KUKA KRL data list: Up22.dat

&ACCESS RVO1
&REL 340
&COMMENT VW380 HO_Behaelter_rechts
&PARAM EDITMASK = Up999[1-999]
&PARAM TEMPLATE = C:\KRC\Roboter\Template\upvorgabe
&PARAM TPVW_VERSION = 8.3.18
&PARAM DISKPATH = UPs
DEFDAT UP22
; FOLD ;%{H} %MKUKATPVW
; ENDFOLD
; interface to basic routines
 EXT  BAS (BAS_COMMAND  :IN,REAL  :IN )
; interface to VW-standard routines
EXT VW (VW_COMMAND:IN, BOOL: IN, REAL:IN, REAL:IN, REAL:IN, REAL:IN, BOOL :IN, E6POS :IN )
; interface to VW_USER - Call
EXT  VW_USER (VW_USER_CMD :IN,INT :IN,REAL  :IN,REAL  :IN,REAL  :IN,REAL  :IN,REAL  :IN,REAL  :IN,REAL  :IN,REAL  :IN,REAL  :IN,BOOL  :IN)
EXT  VW_USR_R (VW_USER_CMD :IN,INT :IN,REAL  :IN,REAL  :IN,REAL  :IN,REAL  :IN,REAL  :IN,REAL  :IN,REAL  :IN,REAL  :IN,REAL  :IN,BOOL  :IN)
EXT  IBGN (IBGN_COMMAND  :IN,BOOL  :IN,REAL  :IN,REAL  :IN,BOOL  :IN,E6POS  :OUT )
; interface select routine
EXTFCT INT  SELECT (SUBTYPE  :IN,INT  :IN,BOOL  :IN,ARI_TYP  :IN,INT  :IN,BOOL_TYP  :IN,INT  :IN,BOOL  :IN)
INT VW_NEXT_FREE = 22
INT VW_NFREE_SPS = 22
INT VW_MAX_SPS = 122
DECL VW_MPARA_TYP P1_D = {TOOL_NO 11,BASE_NO 0,VB 100,VE 0,ACC 100,TRG_TIME 0,MOVE_TYPE #PTP_MOTION}
DECL E6POS P1 = {X 556.5872, Y 1169.977, Z 573.7128, A 30.0, B -0.000000112, C -180.0, S 2, T 3 , E1 0.0, E2 0.0, E3 0.0, E4 0.0, E5 0.0, E6 0.0}
DECL VW_MPARA_TYP P2_D = {TOOL_NO 11,BASE_NO 0,VB 100,VE 100,ACC 100,TRG_TIME 0,MOVE_TYPE #PTP_MOTION}
DECL E6POS P2 = {X 556.5872, Y 1169.977, Z 573.7128, A 30.0, B -0.000000112, C -180.0, S 2, T 3 , E1 0.0, E2 0.0, E3 0.0, E4 0.0, E5 0.0, E6 0.0}
DECL VW_MPARA_TYP P3_D = {TOOL_NO 11,BASE_NO 0,VB 250,VE 50,ACC 100,TRG_TIME 0,MOVE_TYPE #GLUE_MOTION}
DECL E6POS P3 = {X 534.301, Y 1168.777, Z 569.688, A 30.0, B -0.000000111, C -180.0, S 2, T 3 , E1 0.0, E2 0.0, E3 0.0, E4 0.0, E5 0.0, E6 0.0}
DECL VW_MPARA_TYP P4_D = {TOOL_NO 11,BASE_NO 0,VB 250,VE 50,ACC 50,TRG_TIME 0,MOVE_TYPE #GLUE_MOTION}
DECL E6POS P4 = {X 491.0204, Y 1166.447, Z 561.8719, A 30.0, B -0.000000109, C -180.0, S 2, T 3 , E1 0.0, E2 0.0, E3 0.0, E4 0.0, E5 0.0, E6 0.0}
DECL VW_MPARA_TYP P5_D = {TOOL_NO 11,BASE_NO 0,VB 250,VE 50,ACC 100,TRG_TIME 0,MOVE_TYPE #GLUE_MOTION}
DECL E6POS P5 = {X 384.2884, Y 1184.738, Z 561.8702, A 30.0, B -0.000000115, C -180.0, S 2, T 3 , E1 0.0, E2 0.0, E3 0.0, E4 0.0, E5 0.0, E6 0.0}
DECL VW_MPARA_TYP P6_D = {TOOL_NO 11,BASE_NO 0,VB 100,VE 100,ACC 100,TRG_TIME 0,MOVE_TYPE #PTP_MOTION}
DECL E6POS P6 = {X 384.2884, Y 1184.738, Z 579.3517, A 30.0, B -0.000000117, C -180.0, S 2, T 3 , E1 0.0, E2 0.0, E3 0.0, E4 0.0, E5 0.0, E6 0.0}
DECL VW_MPARA_TYP P7_D = {TOOL_NO 11,BASE_NO 0,VB 100,VE 100,ACC 100,TRG_TIME 0,MOVE_TYPE #PTP_MOTION}
DECL E6POS P7 = {X 442.7902, Y 1762.65, Z 1887.477, A 21.55133, B 0.189589, C -113.1255, S 2, T 11 , E1 0.0, E2 0.0, E3 0.0, E4 0.0, E5 0.0, E6 0.0}
DECL VW_MPARA_TYP P8_D = {TOOL_NO 11,BASE_NO 0,VB 100,VE 100,ACC 100,TRG_TIME 0,MOVE_TYPE #PTP_MOTION}
DECL E6POS P8 = {X 1389.959, Y -964.325, Z 1804.324, A -67.67957, B -11.13691, C -126.3533, S 2, T 10 , E1 0.0, E2 0.0, E3 0.0, E4 0.0, E5 0.0, E6 0.0}
DECL VW_MPARA_TYP P9_D = {TOOL_NO 11,BASE_NO 0,VB 100,VE 100,ACC 100,TRG_TIME 0,MOVE_TYPE #PTP_MOTION}
DECL E6POS P9 = {X 591.5993, Y -1509.546, Z 1783.347, A -93.98762, B -12.54844, C -129.5027, S 2, T 10 , E1 0.0, E2 0.0, E3 0.0, E4 0.0, E5 0.0, E6 0.0}
DECL VW_MPARA_TYP P10_D = {TOOL_NO 11,BASE_NO 0,VB 100,VE 100,ACC 100,TRG_TIME 0,MOVE_TYPE #PTP_MOTION}
DECL E6POS P10 = {X 728.618, Y -2376.885, Z 1201.539, A -58.74597, B -24.21727, C -160.5654, S 2, T 10 , E1 0.0, E2 0.0, E3 0.0, E4 0.0, E5 0.0, E6 0.0}
DECL VW_MPARA_TYP P11_D = {TOOL_NO 11,BASE_NO 0,VB 100,VE 100,ACC 100,TRG_TIME 0,MOVE_TYPE #PTP_MOTION}
DECL E6POS P11 = {X 766.4468, Y -2285.862, Z 695.4633, A -38.81029, B -15.174, C -172.4056, S 2, T 10 , E1 0.0, E2 0.0, E3 0.0, E4 0.0, E5 0.0, E6 0.0}
DECL VW_MPARA_TYP P12_D = {TOOL_NO 11,BASE_NO 0,VB 100,VE 0,ACC 100,TRG_TIME 0,MOVE_TYPE #PTP_MOTION}
DECL E6POS P12 = {X 943.1863, Y -1916.042, Z -31.12993, A 2.288836, B 4.706026, C 179.8932, S 2, T 2 , E1 0.0, E2 0.0, E3 0.0, E4 0.0, E5 0.0, E6 0.0}
DECL VW_MPARA_TYP P13_D = {TOOL_NO 11,BASE_NO 3,VB 400,VE 0,ACC 100,TRG_TIME 0,MOVE_TYPE #PATH_MOTION}
DECL E6POS P13 = {X 933.1863, Y -1926.042, Z -41.12993, A 2.288836, B 4.706026, C 179.8932, S 2, T 2 , E1 0.0, E2 0.0, E3 0.0, E4 0.0, E5 0.0, E6 0.0}
DECL VW_MPARA_TYP P14_D = {TOOL_NO 11,BASE_NO 3,VB 400,VE 0,ACC 100,TRG_TIME 0,MOVE_TYPE #PATH_MOTION}
DECL E6POS P14 = {X 2108.789, Y -1906.117, Z -41.1298, A 2.288836, B 4.706027, C 179.8932, S 2, T 2 , E1 0.0, E2 0.0, E3 0.0, E4 0.0, E5 0.0, E6 0.0}
DECL VW_MPARA_TYP P15_D = {TOOL_NO 11,BASE_NO 31,VB 50,VE 100,ACC 100,TRG_TIME 5,MOVE_TYPE #PATH_MOTION}
DECL E6POS P15 = {X -4.24402, Y -0.068859, Z -32.50428, A -2.374263, B 2.921568, C -0.834978, S 2, T 2 , E1 0.0, E2 0.0, E3 0.0, E4 0.0, E5 0.0, E6 0.0}
DECL VW_MPARA_TYP P16_D = {TOOL_NO 11,BASE_NO 31,VB 400,VE 100,ACC 100,TRG_TIME 0,MOVE_TYPE #PATH_MOTION}
DECL E6POS P16 = {X -140.7073, Y -18.48613, Z -69.41855, A -14.37901, B -0.121227, C -1.174702, S 2, T 2 , E1 0.0, E2 0.0, E3 0.0, E4 0.0, E5 0.0, E6 0.0}
DECL VW_MPARA_TYP P17_D = {TOOL_NO 11,BASE_NO 31,VB 400,VE 100,ACC 100,TRG_TIME 0,MOVE_TYPE #PATH_MOTION}
DECL E6POS P17 = {X -150.9838, Y -5.435208, Z -101.0786, A -16.92104, B 0.801226, C -3.417933, S 2, T 2 , E1 0.0, E2 0.0, E3 0.0, E4 0.0, E5 0.0, E6 0.0}
DECL VW_MPARA_TYP P18_D = {TOOL_NO 11,BASE_NO 3,VB 1500,VE 0,ACC 100,TRG_TIME 0,MOVE_TYPE #PATH_MOTION}
DECL E6POS P18 = {X 823.1923, Y -1921.08, Z 71.98488, A 19.24675, B 3.732093, C 177.8513, S 2, T 2 , E1 0.0, E2 0.0, E3 0.0, E4 0.0, E5 0.0, E6 0.0}
DECL VW_MPARA_TYP P19_D = {TOOL_NO 11,BASE_NO 0,VB 100,VE 100,ACC 100,TRG_TIME 0,MOVE_TYPE #PTP_MOTION}
DECL E6POS P19 = {X 653.6893, Y -1905.457, Z 205.6659, A 22.00126, B 3.681432, C -179.4122, S 2, T 2 , E1 0.0, E2 0.0, E3 0.0, E4 0.0, E5 0.0, E6 0.0}
DECL VW_MPARA_TYP P20_D = {TOOL_NO 11,BASE_NO 0,VB 100,VE 100,ACC 100,TRG_TIME 0,MOVE_TYPE #PTP_MOTION}
DECL E6POS P20 = {X 590.098, Y -2159.726, Z 863.7047, A -34.26128, B -9.803282, C 164.3542, S 2, T 2 , E1 0.0, E2 0.0, E3 0.0, E4 0.0, E5 0.0, E6 0.0}
DECL VW_MPARA_TYP P21_D = {TOOL_NO 11,BASE_NO 0,VB 100,VE 0,ACC 100,TRG_TIME 0,MOVE_TYPE #PTP_MOTION}
DECL E6POS P21 = {X 856.7742, Y -895.0887, Z 803.2177, A 3.272736, B 3.014662, C 179.9311, S 2, T 2 , E1 0.0, E2 0.0, E3 0.0, E4 0.0, E5 0.0, E6 0.0}
ENDDAT
